(* Logix 5000 project; controller Reto2 vendor 1 type 14 code 156 rev 30.11; software revision 30.00 *)

TASK MainTask (continuous, watchdog 500 ms) : MainProgram

MODULES
   Local : vendor 1 type 14 code 156 (Compact 0, rev 30.11)
      Digital_IN : 1769-IQ16 (Compact 4, rev 1.1, Input RPI 20 ms)
      Digital_OUT : vendor 1 type 7 code 86 (Compact 5, rev 2.1, Output RPI 20 ms)
      Analog_IN : vendor 1 type 10 code 44 (Compact 2, rev 2.1, Output RPI 80 ms)
      Analog_OUT : vendor 1 type 10 code 48 (Compact 3, rev 1.1, Output RPI 80 ms)
END_MODULES

VAR_GLOBAL   (* controller tags *)
   Any_Pallet : BOOL;
   BOOL_IN_0 : BOOL;   // AUTO
   BOOL_IN_1 : BOOL := 1;   // BOOL AT ENTRY
   BOOL_IN_10 : BOOL;   // PLATE LIMIT
   BOOL_IN_11 : BOOL;   // PUSHER LIMIT
   BOOL_IN_12 : BOOL;   // RESET
   BOOL_IN_13 : BOOL;   // START
   BOOL_IN_14 : BOOL;   // STOP
   BOOL_IN_2 : BOOL;   // CLAMPED
   BOOL_IN_3 : BOOL;   // ELEVATOR MOVING
   BOOL_IN_4 : BOOL := 1;   // EMERGENCY STOP
   BOOL_IN_5 : BOOL;   // FACTORY I/0 (RUNNING)
   BOOL_IN_6 : BOOL;   // MANUAL
   BOOL_IN_7 : BOOL := 1;   // PALLET AT ENTRY
   BOOL_IN_8 : BOOL := 1;   // PALLET AT EXIT
   BOOL_IN_9 : BOOL;   // PALLET LOADED
   BOOL_OUT_0 : BOOL;   // BOX FEEDER
   BOOL_OUT_1 : BOOL;   // CLAMP
   BOOL_OUT_10 : BOOL;   // PUSH
   BOOL_OUT_11 : BOOL;   // TURN
   BOOL_OUT_12 : BOOL;   // WARNING LIGHT
   BOOL_OUT_2 : BOOL;   // ELEVATOR DOWN
   BOOL_OUT_3 : BOOL;   // ELEVATOR UP
   BOOL_OUT_4 : BOOL;   // EXIT CONVEYOR
   BOOL_OUT_5 : BOOL;   // LOAD BELT
   BOOL_OUT_6 : BOOL;   // LOAD PALLET
   BOOL_OUT_7 : BOOL;   // MOVE TO LIMIT
   BOOL_OUT_8 : BOOL;   // OPEN PLATE
   BOOL_OUT_9 : BOOL;   // PALLET FEEDER
   Contador1 : COUNTER := (PRE := 2, CU := 1);
   Contador2 : COUNTER := (PRE := 3, ACC := 1, CU := 1);
   Contador3 : COUNTER := (PRE := 3, CU := 1);
   Contador4 : COUNTER := (PRE := 2, CU := 1);
   Contador5 : COUNTER := (PRE := 3);
   contador6 : COUNTER;
   Contador7 : COUNTER;
   CONTRAER_DE : ALIAS FOR Local:5:O.Data.5;   // Piston Doble efecto Contraer Fisico
   ctu3 : COUNTER := (PRE := 1);
   EXTENDER_DE : ALIAS FOR Local:5:O.Data.4;   // Piston Doble efecto Extender Fisico
   EXTENDER_SE : ALIAS FOR Local:5:O.Data.6;   // Piston Simple Efecto Fisico
   FLOAT_OUT_0 : REAL;
   INT_OUT_0 : DINT;   // CONTADOR CAJAS
   INT_OUT_1 : DINT;   // CONTADOR PALLET
   MOTORAC_FISICO : ALIAS FOR Local:5:O.Data.0;   // Motor AC Fisico
   osb3 : BOOL;
   osb4 : BOOL;
   osb5 : BOOL;
   osb6 : BOOL;
   osb7 : BOOL;
   osb8 : BOOL;
   osf1 : BOOL;
   osf11 : BOOL;
   osf2 : BOOL;
   osf3 : BOOL;
   osf4 : BOOL;
   osf6 : BOOL;
   osf8 : BOOL;
   osr3 : BOOL;
   osr5 : BOOL;
   osr7 : BOOL;
   Pallet_in_Position : BOOL;
   Pallet_Ready_Down : BOOL;
   Pallet_Ready_Up : BOOL;
   Palletizado_finished : BOOL;
   q : BOOL := 1;
   q2 : BOOL;
   q3 : BOOL;
   q5 : BOOL;
   q6 : TIMER := (PRE := 1000);
   sb1 : BOOL;
   sb2 : BOOL;
   st3 : BOOL;
   START_FISICO : ALIAS FOR Local:4:I.Data.1;   // Boton verde Fisico
   START_SCADA : BOOL;   // Boton verde SCADA
   STOP_FISICO : ALIAS FOR Local:4:I.Data.0;   // Boton rojo Fisico
   STOP_SCADA : BOOL;   // Boton rojo SCADA
   Temp : BOOL;
   timer1 : TIMER := (PRE := 3000);
   timer2 : TIMER := (PRE := 600);
   Timer3 : TIMER := (PRE := 200);
   timer4 : TIMER := (PRE := 1000);
   timer5 : TIMER := (PRE := 1000);
   timer6 : TIMER := (PRE := 500);
   timer7 : TIMER := (PRE := 2000);
   TON5 : TIMER := (PRE := 100);
   V_VARIADOR : DINT;
   VARIADOR : ALIAS FOR Local:3:O.Ch0Data;
   VEL_VARIADOR : DINT;
   X : BOOL;
   Y : BOOL;
END_VAR

PROGRAM MainProgram   (* main routine MainRoutine *)

ROUTINE Acomodar_Cajas   (* ladder *)
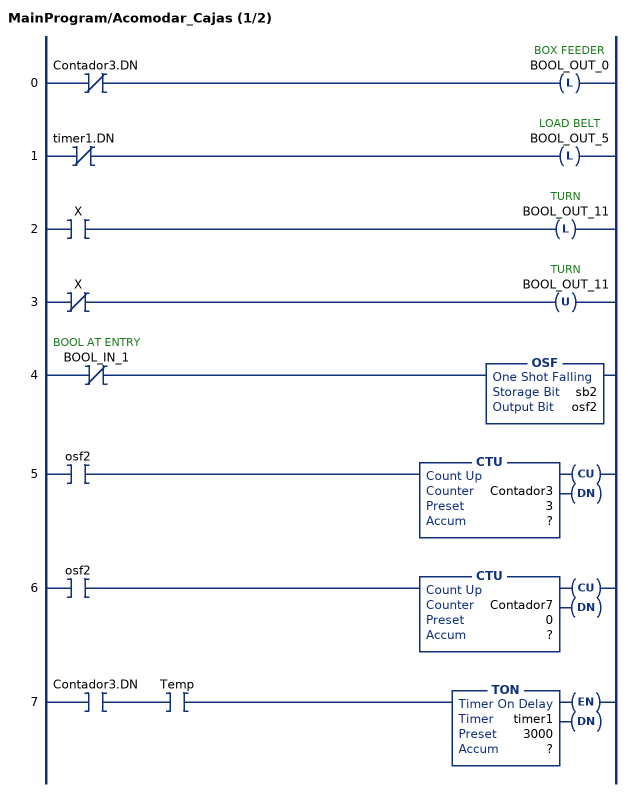
   0: XIO(Contador3.DN)OTL(BOOL_OUT_0);
   1: XIO(timer1.DN)OTL(BOOL_OUT_5);
   2: XIC(X)OTL(BOOL_OUT_11);
   3: XIO(X)OTU(BOOL_OUT_11);
   4: XIO(BOOL_IN_1)OSF(sb2,osf2);
   5: XIC(osf2)CTU(Contador3,?,?);
   6: XIC(osf2)CTU(Contador7,?,?);
   7: XIC(Contador3.DN)XIC(Temp)TON(timer1,?,?);
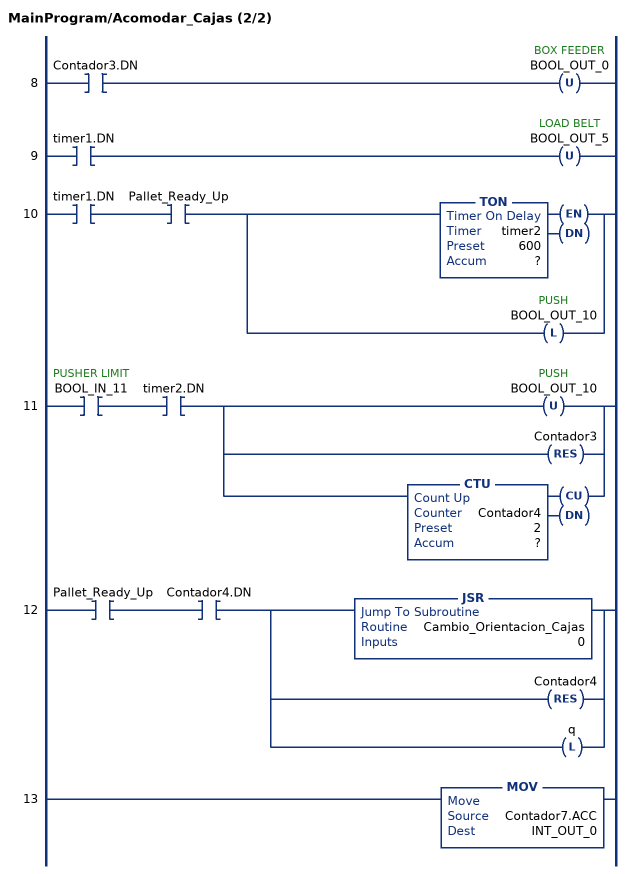
   8: XIC(Contador3.DN)OTU(BOOL_OUT_0);
   9: XIC(timer1.DN)OTU(BOOL_OUT_5);
   10: XIC(timer1.DN)XIC(Pallet_Ready_Up)[TON(timer2,?,?) ,OTL(BOOL_OUT_10) ];
   11: XIC(BOOL_IN_11)XIC(timer2.DN)[[OTU(BOOL_OUT_10) ,RES(Contador3) ] ,CTU(Contador4,?,?) ];
   12: XIC(Pallet_Ready_Up)XIC(Contador4.DN)[[JSR(Cambio_Orientacion_Cajas,0) ,RES(Contador4) ] ,OTL(q) ];
   13: MOV(Contador7.ACC,INT_OUT_0);
END_ROUTINE

ROUTINE Acomodar_Pallet   (* ladder *)
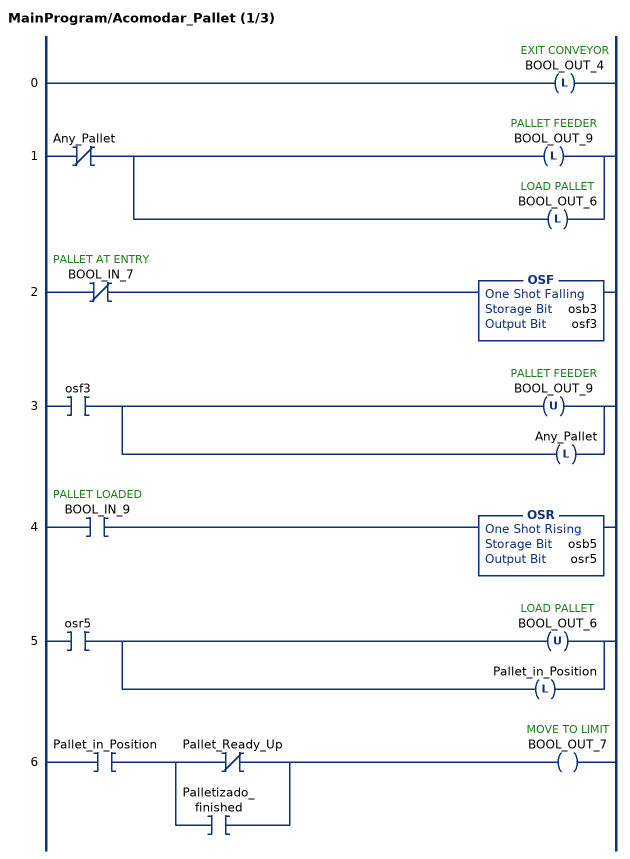
   0: OTL(BOOL_OUT_4);
   1: XIO(Any_Pallet)[OTL(BOOL_OUT_9) ,OTL(BOOL_OUT_6) ];
   2: XIO(BOOL_IN_7)OSF(osb3,osf3);
   3: XIC(osf3)[OTU(BOOL_OUT_9) ,OTL(Any_Pallet) ];
   4: XIC(BOOL_IN_9)OSR(osb5,osr5);
   5: XIC(osr5)[OTU(BOOL_OUT_6) ,OTL(Pallet_in_Position) ];
   6: XIC(Pallet_in_Position)[XIO(Pallet_Ready_Up) ,XIC(Palletizado_finished) ]OTE(BOOL_OUT_7);
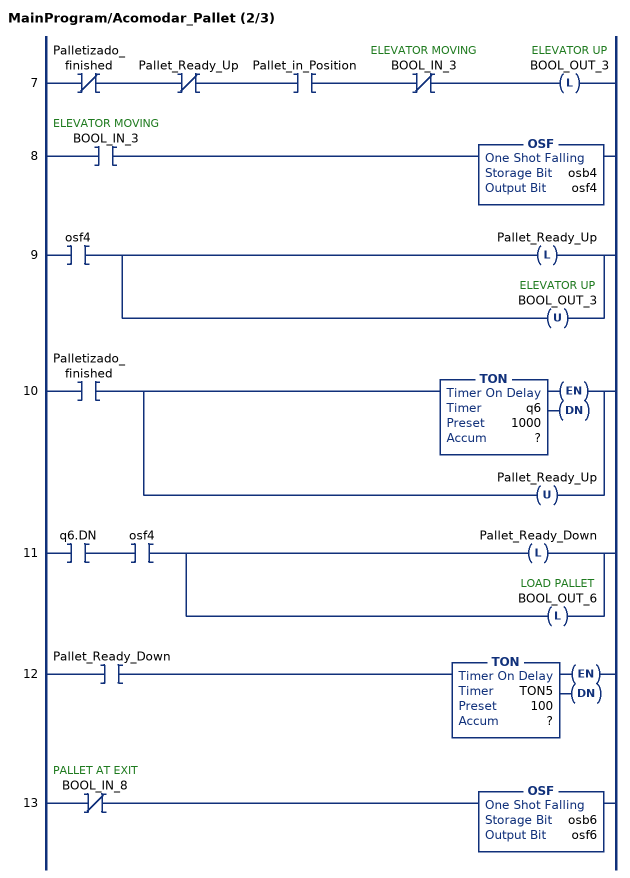
   7: XIO(Palletizado_finished)XIO(Pallet_Ready_Up)XIC(Pallet_in_Position)XIO(BOOL_IN_3)OTL(BOOL_OUT_3);
   8: XIC(BOOL_IN_3)OSF(osb4,osf4);
   9: XIC(osf4)[OTL(Pallet_Ready_Up) ,OTU(BOOL_OUT_3) ];
   10: XIC(Palletizado_finished)[TON(q6,?,?) ,OTU(Pallet_Ready_Up) ];
   11: XIC(q6.DN)XIC(osf4)[OTL(Pallet_Ready_Down) ,OTL(BOOL_OUT_6) ];
   12: XIC(Pallet_Ready_Down)TON(TON5,?,?);
   13: XIO(BOOL_IN_8)OSF(osb6,osf6);
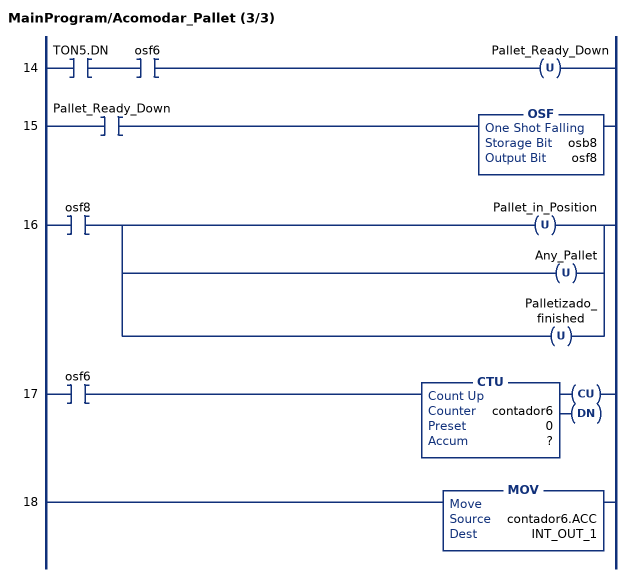
   14: XIC(TON5.DN)XIC(osf6)OTU(Pallet_Ready_Down);
   15: XIC(Pallet_Ready_Down)OSF(osb8,osf8);
   16: XIC(osf8)[OTU(Pallet_in_Position) ,[OTU(Any_Pallet) ,OTU(Palletizado_finished) ] ];
   17: XIC(osf6)CTU(contador6,?,?);
   18: MOV(contador6.ACC,INT_OUT_1);
END_ROUTINE

ROUTINE Cambio_Orientacion_Cajas   (* structured text *)
   if X or not BOOL_IN_5 then
   	X := 0;
   	Contador3.PRE := 2;
   	Contador4.PRE := 3;
   else
   	X := 1;
   	Contador3.PRE := 3;
   	Contador4.PRE := 2;
   end_if;
END_ROUTINE

ROUTINE Conexion_Fisica   (* ladder *)
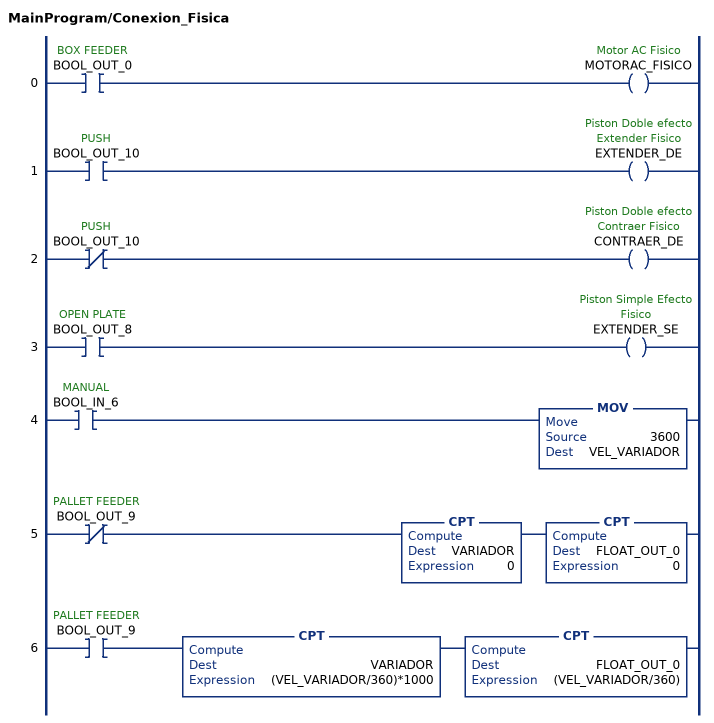
   0: XIC(BOOL_OUT_0)OTE(MOTORAC_FISICO);
   1: XIC(BOOL_OUT_10)OTE(EXTENDER_DE);
   2: XIO(BOOL_OUT_10)OTE(CONTRAER_DE);
   3: XIC(BOOL_OUT_8)OTE(EXTENDER_SE);
   4: XIC(BOOL_IN_6)MOV(3600,VEL_VARIADOR);
   5: XIO(BOOL_OUT_9)CPT(VARIADOR,0)CPT(FLOAT_OUT_0,0);
   6: XIC(BOOL_OUT_9)CPT(VARIADOR,(VEL_VARIADOR/360)*1000)CPT(FLOAT_OUT_0,(VEL_VARIADOR/360));
END_ROUTINE

ROUTINE Inicialization   (* structured text *)
   if not(BOOL_IN_5) then
   	BOOL_OUT_0:=0;
   	BOOL_OUT_1:=0;
   	BOOL_OUT_2:=0;
   	BOOL_OUT_3:=0;
   	BOOL_OUT_4:=0;
   	BOOL_OUT_5:=0;
   	BOOL_OUT_6:=0;
   	BOOL_OUT_7:=0;
   	BOOL_OUT_8:=0;
   	BOOL_OUT_9:=0;
   	BOOL_OUT_10:=0;
   	BOOL_OUT_11:=0;
   	BOOL_OUT_12:=0;
   
   	Palletizado_finished:=0;
   	Pallet_Ready_Up:=0;
   	Pallet_Ready_Down:=0;
   	Pallet_in_Position:=0;
   	Any_Pallet:=0;
   
   	Temp:=0;
   
   	q:=0;
   	q2:=0;
   	q3:=0;
   	q5:=0;
   
   	JSR(Parada);
   	JSR(Reset);
   	JSR(Cambio_Orientacion_Cajas);
   end_if;
END_ROUTINE

ROUTINE MainRoutine   (* ladder *)
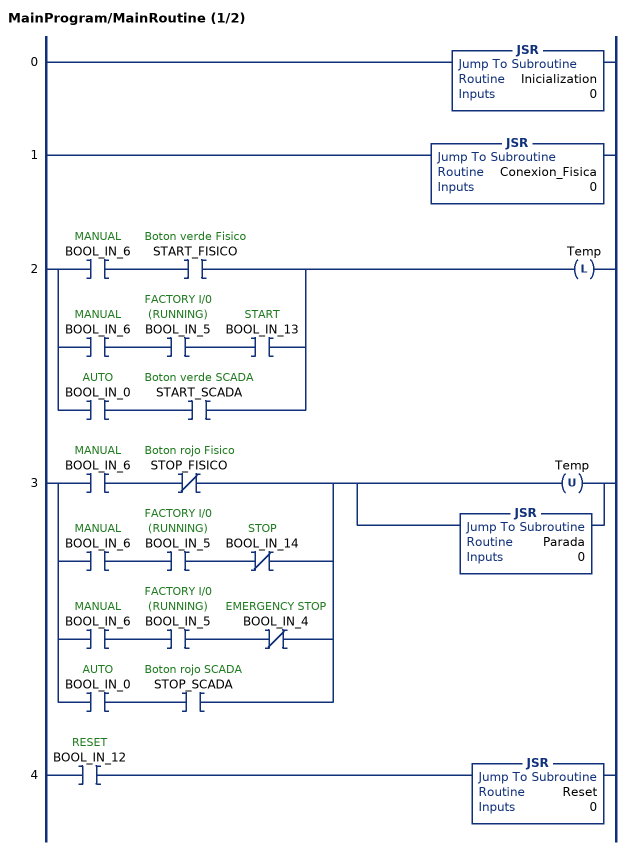
   0: JSR(Inicialization,0);
   1: JSR(Conexion_Fisica,0);
   2: [XIC(BOOL_IN_6) XIC(START_FISICO) ,[XIC(BOOL_IN_6) XIC(BOOL_IN_5) XIC(BOOL_IN_13) ,XIC(BOOL_IN_0) XIC(START_SCADA) ] ]OTL(Temp);
   3: [XIC(BOOL_IN_6) XIO(STOP_FISICO) ,[[XIC(BOOL_IN_6) XIC(BOOL_IN_5) XIO(BOOL_IN_14) ,XIC(BOOL_IN_6) XIC(BOOL_IN_5) XIO(BOOL_IN_4) ] ,XIC(BOOL_IN_0) XIC(STOP_SCADA) ] ][OTU(Temp) ,JSR(Parada,0) ];
   4: XIC(BOOL_IN_12)JSR(Reset,0);
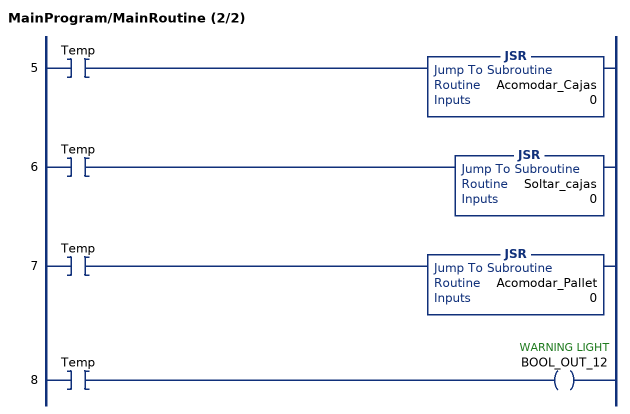
   5: XIC(Temp)JSR(Acomodar_Cajas,0);
   6: XIC(Temp)JSR(Soltar_cajas,0);
   7: XIC(Temp)JSR(Acomodar_Pallet,0);
   8: XIC(Temp)OTE(BOOL_OUT_12);
END_ROUTINE

ROUTINE Parada   (* ladder *)
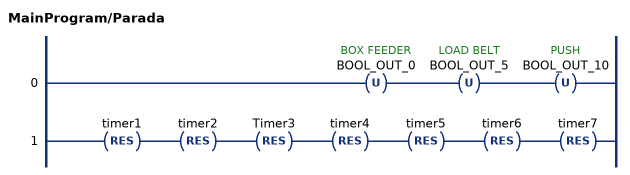
   0: OTU(BOOL_OUT_0)OTU(BOOL_OUT_5)OTU(BOOL_OUT_10);
   1: RES(timer1)RES(timer2)RES(Timer3)RES(timer4)RES(timer5)RES(timer6)RES(timer7);
END_ROUTINE

ROUTINE Reset   (* ladder *)
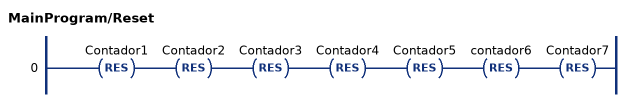
   0: RES(Contador1)RES(Contador2)RES(Contador3)RES(Contador4)RES(Contador5)RES(contador6)RES(Contador7);
END_ROUTINE

ROUTINE Soltar_cajas   (* ladder *)
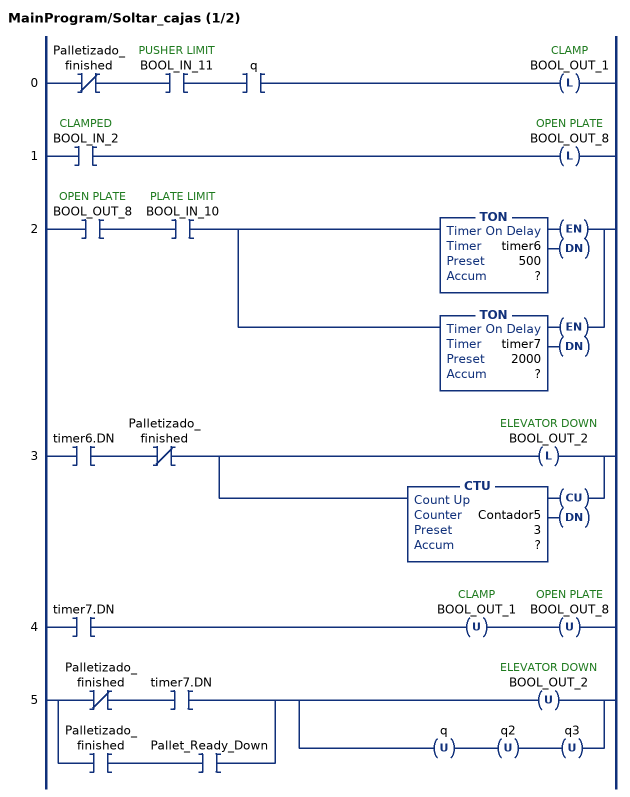
   0: XIO(Palletizado_finished)XIC(BOOL_IN_11)XIC(q)OTL(BOOL_OUT_1);
   1: XIC(BOOL_IN_2)OTL(BOOL_OUT_8);
   2: XIC(BOOL_OUT_8)XIC(BOOL_IN_10)[TON(timer6,?,?) ,TON(timer7,?,?) ];
   3: XIC(timer6.DN)XIO(Palletizado_finished)[OTL(BOOL_OUT_2) ,CTU(Contador5,?,?) ];
   4: XIC(timer7.DN)OTU(BOOL_OUT_1)OTU(BOOL_OUT_8);
   5: [XIO(Palletizado_finished) XIC(timer7.DN) ,XIC(Palletizado_finished) XIC(Pallet_Ready_Down) ][OTU(BOOL_OUT_2) ,OTU(q) OTU(q2) OTU(q3) ];
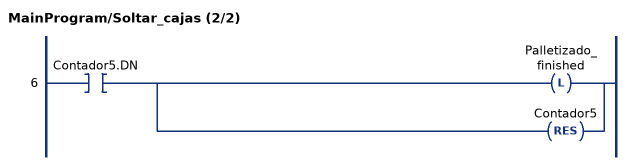
   6: XIC(Contador5.DN)[OTL(Palletizado_finished) ,RES(Contador5) ];
END_ROUTINE
END_PROGRAM
